(* PLC project Unnamed, Unknown Unnamed 1 *)
(* stored: creationDateTime 2023-08-01T21:16:32, modificationDateTime 2023-08-03T14:07:25 *)

PROGRAM main
  VAR
    in : BOOL;
    out : BOOL;
  END_VAR

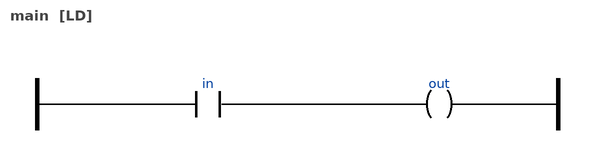
(* LD diagram, written out as Structured Text *)
out := in;
END_PROGRAM

PROGRAM get_temp
  VAR
    I2C_AHT200 : I2C_AHT20;
    sck : INT;
    sda : INT;
    temp : REAL;
  END_VAR

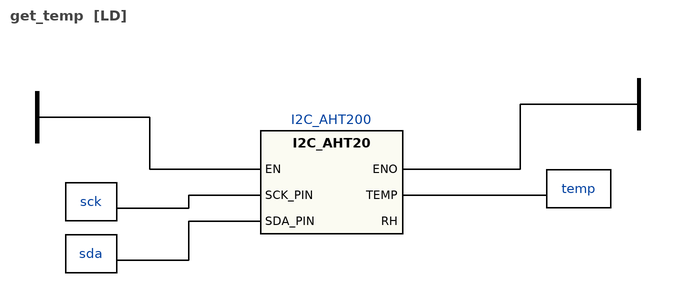
(* LD diagram, written out as Structured Text *)
I2C_AHT200(SCK_PIN := sck, SDA_PIN := sda);
temp := I2C_AHT200.TEMP;
END_PROGRAM

CONFIGURATION Config0
  RESOURCE Res0 ON PLC
    VAR_GLOBAL
      T0 : REAL;
      SCK_PIN : INT := 22;
      SDA_PIN : INT := 21;
    END_VAR
    TASK task0(INTERVAL := T#20ms, PRIORITY := 0);
    TASK task1(INTERVAL := T#1000ms, PRIORITY := 1);
    PROGRAM instance0 WITH task0 : main;
    PROGRAM instance1 WITH task0 : get_temp;
  END_RESOURCE
END_CONFIGURATION
